FUNCTION_BLOCK FB_System_SHZ_350
VAR_INPUT
	Betrieb_Anford_auto		: BOOL;
	Regelung_Modus_auto		: USINT;
	Regelung_Sollw_auto		: REAL;
	Temp_Aussen				: REAL;
	Temp_Innen				: REAL;
END_VAR
VAR_OUTPUT
END_VAR
VAR
	{attribute 'OPC.UA.DA' := '1'}Steuerung				: ST_System_SHZ_Steuerung;		
	{attribute 'OPC.UA.DA' := '1'}Stellwert					: ST_System_SHZ_Stellwert;	
	{attribute 'OPC.UA.DA' := '1'}Zustand					: ST_System_SHZ_Zustand;	
	{attribute 'OPC.UA.DA' := '1'}Parameter				: ST_System_SHZ_Parameter;		

	Pumpe_350				: FB_PU;
	Regelventil_350			: FB_RV;

	Zustandscheck			: FB_System_SHZ_Zustandscheck;
	Logik					: FB_System_SHZ_Logik;
	Ablaufsteuerung			: FB_System_SHZ_Ablaufsteuerung;
	Sollwertscheck			: FB_System_SHZ_Sollwertscheck;
	Regelung				: FB_System_SHZ_Regelung;
	Stellwertscheck			: FB_System_SHZ_Stellwertscheck;

	Test_Temp_Aussen		: USINT;
	Test_Wetter_Temperatur: REAL;
END_VAR

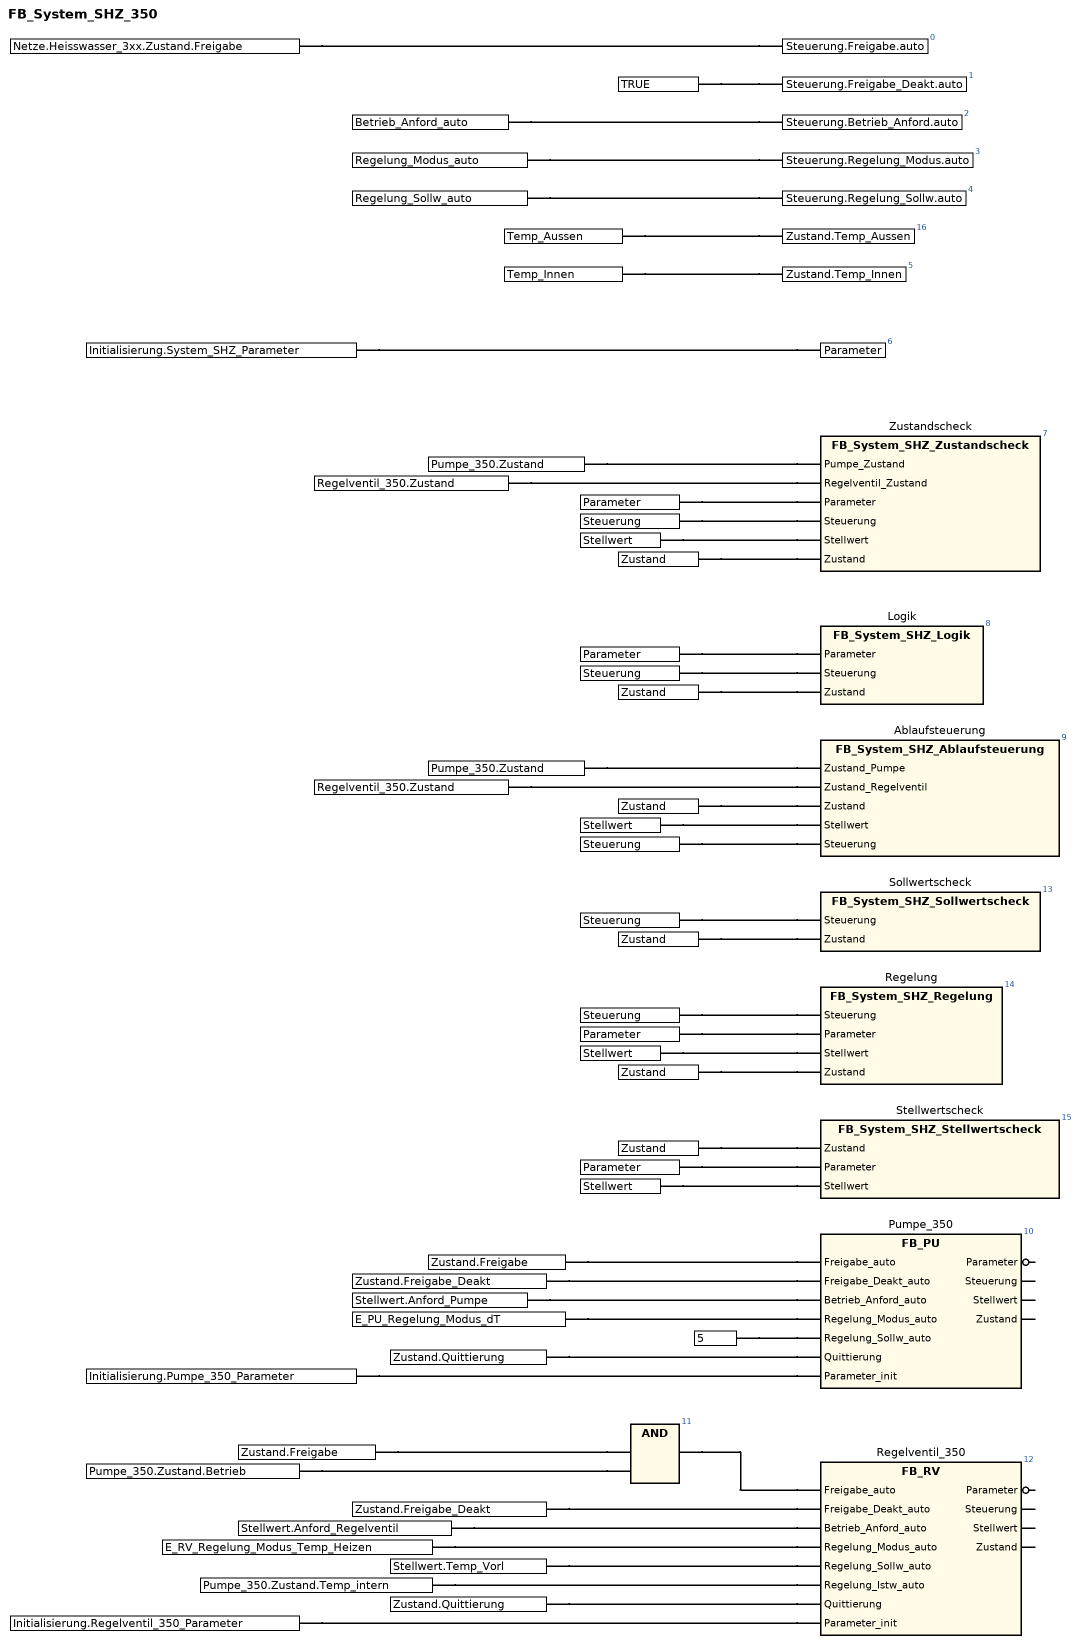
Steuerung.Freigabe.auto := Netze.Heisswasser_3xx.Zustand.Freigabe;
Steuerung.Freigabe_Deakt.auto := TRUE;
Steuerung.Betrieb_Anford.auto := Betrieb_Anford_auto;
Steuerung.Regelung_Modus.auto := Regelung_Modus_auto;
Steuerung.Regelung_Sollw.auto := Regelung_Sollw_auto;
Zustand.Temp_Innen := Temp_Innen;
Parameter := Initialisierung.System_SHZ_Parameter;
Zustandscheck(
    Pumpe_Zustand := Pumpe_350.Zustand,
    Regelventil_Zustand := Regelventil_350.Zustand,
    Parameter := Parameter,
    Steuerung := Steuerung,
    Stellwert := Stellwert,
    Zustand := Zustand); // FB_System_SHZ_Zustandscheck
Logik(Parameter := Parameter, Steuerung := Steuerung, Zustand := Zustand); // FB_System_SHZ_Logik
Ablaufsteuerung(
    Zustand_Pumpe := Pumpe_350.Zustand,
    Zustand_Regelventil := Regelventil_350.Zustand,
    Zustand := Zustand,
    Stellwert := Stellwert,
    Steuerung := Steuerung); // FB_System_SHZ_Ablaufsteuerung
Pumpe_350(
    Freigabe_auto := Zustand.Freigabe,
    Freigabe_Deakt_auto := Zustand.Freigabe_Deakt,
    Betrieb_Anford_auto := Stellwert.Anford_Pumpe,
    Regelung_Modus_auto := E_PU_Regelung_Modus_dT,
    Regelung_Sollw_auto := 5,
    Quittierung := Zustand.Quittierung,
    Parameter_init := Initialisierung.Pumpe_350_Parameter); // FB_PU
Regelventil_350(
    Freigabe_auto := Zustand.Freigabe AND Pumpe_350.Zustand.Betrieb,
    Freigabe_Deakt_auto := Zustand.Freigabe_Deakt,
    Betrieb_Anford_auto := Stellwert.Anford_Regelventil,
    Regelung_Modus_auto := E_RV_Regelung_Modus_Temp_Heizen,
    Regelung_Sollw_auto := Stellwert.Temp_Vorl,
    Regelung_Istw_auto := Pumpe_350.Zustand.Temp_intern,
    Quittierung := Zustand.Quittierung,
    Parameter_init := Initialisierung.Regelventil_350_Parameter); // FB_RV
Sollwertscheck(Steuerung := Steuerung, Zustand := Zustand); // FB_System_SHZ_Sollwertscheck
Regelung(Steuerung := Steuerung, Parameter := Parameter, Stellwert := Stellwert, Zustand := Zustand); // FB_System_SHZ_Regelung
Stellwertscheck(Zustand := Zustand, Parameter := Parameter, Stellwert := Stellwert); // FB_System_SHZ_Stellwertscheck
Zustand.Temp_Aussen := Temp_Aussen;

END_FUNCTION_BLOCK

(* stored: Version 1.1.0.1, ProductVersion 3.1.4024.9
   POU FB_System_SHZ_350: Id {8bd4dfa4-30bf-45d9-9764-ac133b24a0be}, SpecialFunc None *)
